Yaskawa INFORM job: POS_TEST7.JBI

/JOB
//NAME POS_TEST7
//POS
///NPOS 2,0,0,12,0,0
///POSTYPE BASE
///RECTAN
C00000=2000.000,-300.000,-450.000,180.0000,-90.0000,0.0000
C00001=2000.000,350.000,-450.000,180.0000,-90.0000,0.0000
///POSTYPE BASE
///RECTAN
P00030=1000.000,500.000,-500.000,0.0000,0.0000,0.0000
P00031=1100.000,-500.000,-400.000,0.0000,0.0000,0.0000
P00032=1000.000,400.000,-400.000,0.0000,0.0000,0.0000
P00033=1100.000,-400.000,-300.000,0.0000,0.0000,0.0000
P00034=1000.000,300.000,-300.000,0.0000,0.0000,0.0000
P00035=1100.000,-300.000,-200.000,0.0000,0.0000,0.0000
P00036=1000.000,200.000,-200.000,0.0000,0.0000,0.0000
P00037=1100.000,-200.000,-100.000,0.0000,0.0000,0.0000
P00038=1000.000,100.000,-100.000,0.0000,0.0000,0.0000
P00039=1100.000,-100.000,0.000,0.0000,0.0000,0.0000
P00040=1000.000,50.000,0.000,0.0000,0.0000,0.0000
P00041=1100.000,-50.000,50.000,0.0000,0.0000,0.0000
//INST
///DATE 2023/06/06 15:44
///ATTR SC,RW,RJ
////FRAME BASE
///GROUP1 RB1
NOP
MOVJ P009 VJ=15.00
SET I001 85
SET I002 218
SET I003 29
FOR I000 START= 13 TO 18
	SET D000 65
	SETPRM KIND=5 PRMNO=I000 D000
	SET D000 1
	ADD I001 2
	SETPRM KIND=5 PRMNO=I001 D000
	INC I003
	GETE D000 P[I003] (1)
	GETE D001 P[I003] (2)
	GETE D002 P[I003] (3)
	ADD I002 6
	SETPRM KIND=6 PRMNO=I002 D000
	INC I002
	SETPRM KIND=6 PRMNO=I002 D001
	INC I002
	SETPRM KIND=6 PRMNO=I002 D002
	INC I003
	GETE D000 P[I003] (1)
	GETE D001 P[I003] (2)
	GETE D002 P[I003] (3)
	ADD I002 6
	SETPRM KIND=6 PRMNO=I002 D000
	INC I002
	SETPRM KIND=6 PRMNO=I002 D001
	INC I002
	SETPRM KIND=6 PRMNO=I002 D002
NEXT I000
MOVJ C000 VJ=12.0
MOVL C001 V=150.0
END
